FUNCTION_BLOCK WeightSensor IMPLEMENTS ITF_AnalogSensor
VAR_INPUT
END_VAR
VAR_OUTPUT
END_VAR
VAR
	AI_WPWeight AT %I* : INT;
END_VAR

PROPERTY Value : INT
GET
Value := AI_WPWeight;
END_GET
END_PROPERTY

END_FUNCTION_BLOCK

(* stored: Version 1.1.0.1
   POU WeightSensor: Id {9c9a8d30-bf02-4b6b-a6ef-1b857fd4298b}, SpecialFunc None
   Property Value: Id {0bc90006-697b-4de8-867b-f25d5aac15d8}
   Get Get: Id {56d0623e-779f-4ef9-8f01-12ead08c35e2} *)
